(* PLC project SL-RP4, OpenPLC SL-RP4 1.0, author OpenPLC Lib Writter *)
(* stored: creationDateTime 2023-04-26T04:54:00, modificationDateTime 2023-04-26T04:54:00 *)

(* Reads the rotary switch position on SL-RP4 when the READ input is triggered. If ERROR is TRUE then an error occurred while trying to read the rotary switch. If ERROR is FALSE, the switch position value will be available on output OUT *)
FUNCTION_BLOCK ROTARY_SWITCH
  VAR_INPUT
    READ : BOOL;  (* READ *)
  END_VAR
  VAR_OUTPUT
    ERROR : BOOL;  (* ERROR *)
    OUT : INT;  (* OUT *)
  END_VAR

  IF READ = TRUE THEN
    OUT := 0;
  END_IF;
END_FUNCTION_BLOCK
